TYPE st_AxisControl :
STRUCT
	Error	  : BOOL;
	ResetAxis : BOOL;
END_STRUCT
END_TYPE

(* stored: Version 1.1.0.1, ProductVersion 3.1.4024.13
   DUT st_AxisControl: Id {2d309f22-6a80-4e66-a996-f3082c26e9c5} *)
